{attribute 'linkalways'} 
{attribute 'no_explicit_call' := 'This FB is a CLASS and must be accessed using methods or properties'}
{attribute 'enable_dynamic_creation'}
FUNCTION_BLOCK StructuredDatatypeAddedEvent EXTENDS Disposable IMPLEMENTS I_StructuredDatatypeAddedEvent
VAR
	_target : I_StructuredDatatype;
END_VAR

METHOD FB_init : BOOL
VAR_INPUT
	bInitRetains : BOOL; // if TRUE, the retain variables are initialized (warm start / cold start)
	bInCopyCode : BOOL;  // if TRUE, the instance afterwards gets moved into the copy code (online change)
	Target : I_StructuredDatatype;
END_VAR
This^._target := Target;
END_METHOD

PROPERTY PUBLIC Target : I_StructuredDatatype
GET
Target := _target;
END_GET
END_PROPERTY

END_FUNCTION_BLOCK

(* stored: Version 1.1.0.1, ProductVersion 3.1.4024.12
   POU StructuredDatatypeAddedEvent: Id {0ec0ed94-ac70-091e-2a39-3d07144b4499}, SpecialFunc None
   Folder Constructor: Id {04007ff5-8822-0e9f-2c43-38df87bcf932}
   Method FB_init: Id {c333b2fb-c430-0e1a-028f-d6eaa7c757db}
   Property Target: Id {f8014708-a376-0d18-2273-894f8cebb0fc}
   Get Get: Id {23963d23-fa2c-0a3d-266b-2523cb1ce3c1} *)
